FUNCTION_BLOCK GET_PLANAR_FACE_START_POINT (* Get planar face start point *)
  (* Standard: 61499-2 *)
  (* Version 1.0, 21-06-12, GASR, Universidade do Estado de Santa Catarina *)
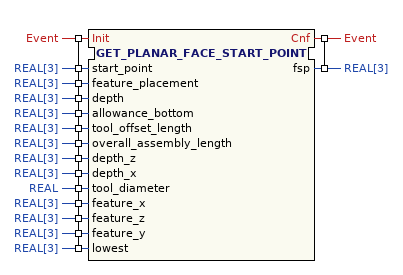
  EVENT_INPUT
    Init WITH start_point, feature_placement, depth, allowance_bottom, tool_offset_length, overall_assembly_length, depth_z, depth_x, tool_diameter, feature_x, feature_z, feature_y, lowest;
  END_EVENT
  EVENT_OUTPUT
    Cnf WITH fsp;
  END_EVENT
  VAR_INPUT
    start_point : ARRAY [0..2] OF REAL; (* Operation start point *)
    feature_placement : ARRAY [0..2] OF REAL; (* Feature local coordinate system origin *)
    depth : ARRAY [0..2] OF REAL; (* Feature depth location *)
    allowance_bottom : ARRAY [0..2] OF REAL; (* Material thickness to be left uncut *)
    tool_offset_length : ARRAY [0..2] OF REAL; (* Tool blade length *)
    overall_assembly_length : ARRAY [0..2] OF REAL; (* Tool length *)
    depth_z : ARRAY [0..2] OF REAL; (* Depth z vector *)
    depth_x : ARRAY [0..2] OF REAL; (* Depth x vector *)
    tool_diameter : REAL;
    feature_x : ARRAY [0..2] OF REAL;
    feature_z : ARRAY [0..2] OF REAL;
    feature_y : ARRAY [0..2] OF REAL;
    lowest : ARRAY [0..2] OF REAL;
  END_VAR
  VAR_OUTPUT
    fsp : ARRAY [0..2] OF REAL; (* feature_start_point *)
  END_VAR
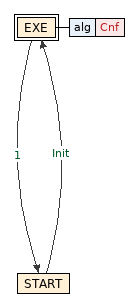
  EC_STATES
    EXE : alg -> Cnf;
    START;
  END_STATES
  EC_TRANSITIONS
    EXE TO START := 1;
    START TO EXE := Init;
  END_TRANSITIONS
  ALGORITHM alg IN Lua:
local max_depth    = depth[3] + allowance_bottom
local blade_length = overall_assembly_length - tool_offset_length
print( 'feature vectors', 'x', feature_x[1], feature_x[2], feature_x[3], 'y', feature_y[1], feature_y[2], feature_y[3] )
print( 'tool_diameter', tool_diameter )
if(( start_point[1] ~= 0 ) and ( start_point[2] ~= 0 ) and ( start_point[3] ~= 0 )) then
    for i = 1, 3 do fsp[i] = start_point[i] end
else
    for i = 1, 3 do fsp[i] = feature_placement[i] end
    fsp[1] = fsp[1] + feature_x[1]*(tool_diameter/2) + feature_y[1]*(tool_diameter/2)
    fsp[2] = fsp[2] + feature_x[2]*(tool_diameter/2) + feature_y[2]*(tool_diameter/2)
    if(( depth_z[1] ~= 0 ) or ( depth_z[2] ~= 0 )) then
        depth_y = { ((depth_z[2]*depth_x[3]) - (depth_x[2]*depth_z[3])),
                    ((depth_z[3]*depth_x[1]) - (depth_x[3]*depth_z[1])),
                    ((depth_z[1]*depth_x[2]) - (depth_x[1]*depth_z[2])) }
        print( 'depth_vectors\n', depth_x[1], depth_x[2], depth_x[3], '\n', depth_y[1], depth_y[2], depth_y[3], '\n', depth_z[1], depth_z[2], depth_z[3], '\n' )
        local t, w
        if( depth_y[1] == 0 ) then
            t = ( fsp[1]/depth_x[1] - depth[1] )
            w = ( fsp[2] - depth[2] - depth_x[2]*t )/depth_y[2]
        elseif( depth_x[1] == 0 ) then
            w = ( fsp[1]/depth_y[1] - depth[2] )
            t = ( fsp[2] - depth[2] - depth_y[2]*w )/depth_y[2]
        else
            t = ( ( fsp[2] - depth_y[2]*fsp[1]/depth_y[1] + depth_y[2]*depth[1]/depth_y[1] - depth[2] )/( depth_x[2] - depth_y[2]*depth_x[2]/depth_y[1] ) )
            w = ( fsp[1] - depth[1] - depth_x[1]*t )/depth_y[1]
        end
        fsp[3] = ( depth_x[3]*t + depth_y[3]*w + depth[3] )
        if( (-blade_length + feature_placement[3]) > lowest[3] ) then
        elseif( blade_length - feature_placement[3] > -fsp[3] ) then
        else
            fsp[3] = -blade_length + feature_placement[3]
        end
    else
        if( blade_length > -max_depth ) then
            fsp[3] = (max_depth + feature_placement[3])
        else
            fsp[3] = (-blade_length + feature_placement[3])
        end
    end
end
print( 'start_point', fsp[1], fsp[2], fsp[3] )
--Check for depth violation
if( math.abs(fsp[3] - feature_placement[3]) > blade_length ) then
    fsp[3] = -blade_length
end
if( math.abs(fsp[3] - feature_placement[3]) > max_depth ) then
    fsp[3] = -max_depth
end
  END_ALGORITHM
END_FUNCTION_BLOCK
